{attribute 'qualified_only'}
// {attribute 'strict'}
TYPE E_OperStateCntrl :
(
	stopped:= 0,
	running:= 1,
	sleeping:= 2,
	overheight:= 3,
	extended := 4,
	extending := 5,
	retracted := 6,
	retracting := 7,
	unknown :=8,
	offline :=9,
	auto := 10,
	manual := 11,
	faulted	:= 12
) INT;
END_TYPE

(* stored: Version 1.1.0.1, ProductVersion 3.1.4024.4
   EnumerationTextList E_OperStateCntrl: Id {0a750aca-6721-4d12-9524-0fd4630f8697} *)
